{attribute addProperty BoxType "EL5122-0000-0016"}
{attribute addProperty Id "ControlAT %Q*Control_2618F9C31620Set_counter_valueAT %Q*UDINT32417"}
{attribute addProperty CRC "1355439456"}
{attribute addProperty SizeInBites "48"}
{attribute addProperty SizeInBytes "6"}
TYPE ENC_Control_Channel_50CA5D60 :
STRUCT
	{attribute addProperty Name "Control"}
	Control AT %Q* : Control_2618F9C3;
	{attribute addProperty Name "Set_counter_value"}
	Set_counter_value AT %Q* : UDINT;
END_STRUCT
END_TYPE

(* stored: Version 1.2.0.0, ProductVersion 3.1.4024.9
   DUT ENC_Control_Channel_50CA5D60: Id {4d5dc952-8715-4a1a-adb9-68b645daa8da} *)
